INTERFACE iSuperActuator

METHOD ErrorHandling : BOOL
VAR_INPUT
END_VAR
END_METHOD

PROPERTY IsError : bool
GET
END_GET
END_PROPERTY

METHOD ResetError : BOOL
VAR_INPUT
END_VAR
END_METHOD

END_INTERFACE

(* stored: Version 1.1.0.1, ProductVersion 3.1.4024.12
   Itf iSuperActuator: Id {7d906433-c242-40bb-a2ff-7356a90c2292}
   Method ErrorHandling: Id {8bb89f97-f6ff-4f7b-9dd5-50a06b17fb3c}
   Property IsError: Id {ebe86b05-d4dc-40ea-9640-96f404873b1e}
   Get Get: Id {392bbca7-14aa-471f-9ef1-45c759f2dbe3}
   Method ResetError: Id {52ca07aa-ba55-4e48-a3d6-2319d7c0005f} *)
